INTERFACE I_ChunkedRequestData EXTENDS I_SessionData

PROPERTY PUBLIC IsComplete : BOOL
GET
END_GET
END_PROPERTY

METHOD PUBLIC TryAddChunkedRequest : BOOL;
VAR_INPUT
	Request : I_Request;
	ChunkSequence : DINT;
END_VAR
END_METHOD

END_INTERFACE

(* stored: Version 1.1.0.1, ProductVersion 3.1.4024.12
   Itf I_ChunkedRequestData: Id {22300d9d-d667-4bc8-b0b3-5a4fa8f36f5d}
   Property IsComplete: Id {dec49cc7-3ada-4338-bf34-8f28fd7fa0b6}
   Get Get: Id {f8c4caa5-5470-45d1-b7a7-46724b7937ce}
   Method TryAddChunkedRequest: Id {ea33a017-e809-4192-9e23-7f6dbb771687} *)
